{attribute 'qualified_only'}
{attribute 'strict'}
{attribute 'to_string'}
TYPE ACTIVITY_RUNNING_STATE :
(
	WORK_IN_PROGRESS := 0,
	WORK_COMPLETED,
	WORK_HALTED
);
END_TYPE

(* stored: Version 1.1.0.1
   DUT ACTIVITY_RUNNING_STATE: Id {24d4d980-d91a-4e70-b1c0-2be206ebd59f} *)
